{attribute 'GeneratedUsingTerminal: KL9999'}
{attribute addProperty BoxType "KL9999"}
{attribute addProperty Description ""}
{attribute addProperty Physics ""}
{attribute addProperty Id "Channel_1AT %Q*Channel_126527430"}
{attribute addProperty CRC "2047911926"}
{attribute addProperty Size "0"}
TYPE KL9999_7A10A7F6 :
STRUCT
	{attribute addProperty Name "Channel_1"}
	Channel_1 : Channel_12652743;
END_STRUCT
END_TYPE

(* stored: Version 1.2.0.0, ProductVersion 3.1.4024.11
   DUT KL9999_7A10A7F6: Id {bef70ada-7928-442a-8024-1ac5c54754e9} *)
